// SIMATIC S7-200 project (STEP 7-Micro/WIN), CPU 224 REL 02.01

ORGANIZATION_BLOCK PRINCIPAL:OB1
TITLE=Uso de Temporizadores, Contadores y Contacto de Transición en PLC S7-200 modelo 224.
BEGIN
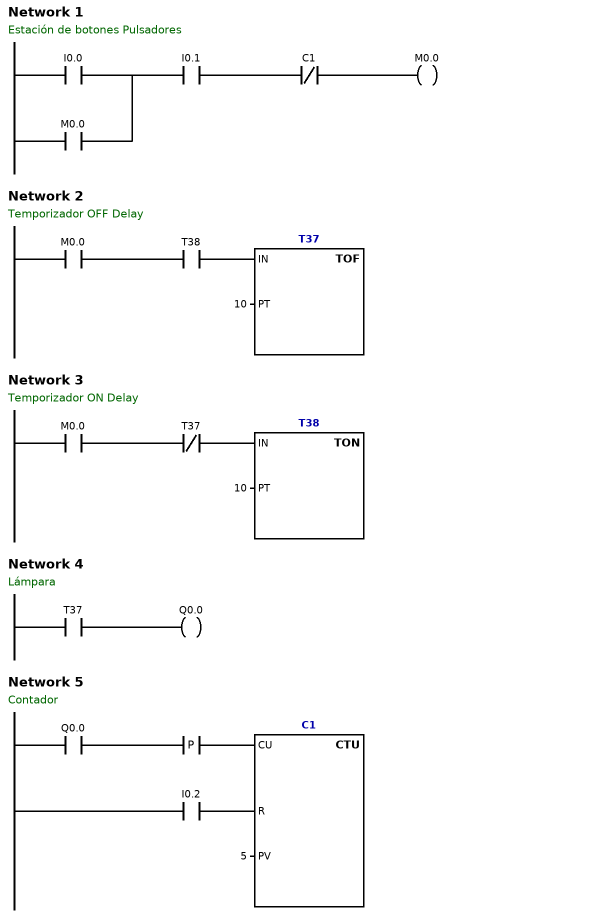
Network 1
// Estación de botones Pulsadores
// (network saved uncompiled; LAD cells follow)
// row 0: c0 -| |- I0.0 v  c1 -| |- I0.1  c2 -|/|- C1  c3 -( ) M0.0
// row 1: c0 -| |- M0.0 ^
Network 2
// Temporizador OFF Delay
// (network saved uncompiled; LAD cells follow)
// row 0: c0 -| |- M0.0  c1 -| |- T38  c2 [TOF T37 IN:=power@row0, PT:=10]
// row 1: c2 [box]
Network 3
// Temporizador ON Delay
// (network saved uncompiled; LAD cells follow)
// row 0: c0 -| |- M0.0  c1 -|/|- T37  c2 [TON T38 IN:=power@row0, PT:=10]
// row 1: c2 [box]
Network 4
// Lámpara
// (network saved uncompiled; LAD cells follow)
// row 0: c0 -| |- T37  c1 -( ) Q0.0
Network 5
// Contador
// (network saved uncompiled; LAD cells follow)
// row 0: c0 -| |- Q0.0  c1 -|P|-  c2 [CTU C1 CU:=power@row0, R:=power@row1, PV:=5]
// row 1: c0 --  c1 -| |- I0.2  c2 [box]
// row 2: c2 [box]
END_ORGANIZATION_BLOCK
